RoboDK station: Assignment 3.rdk

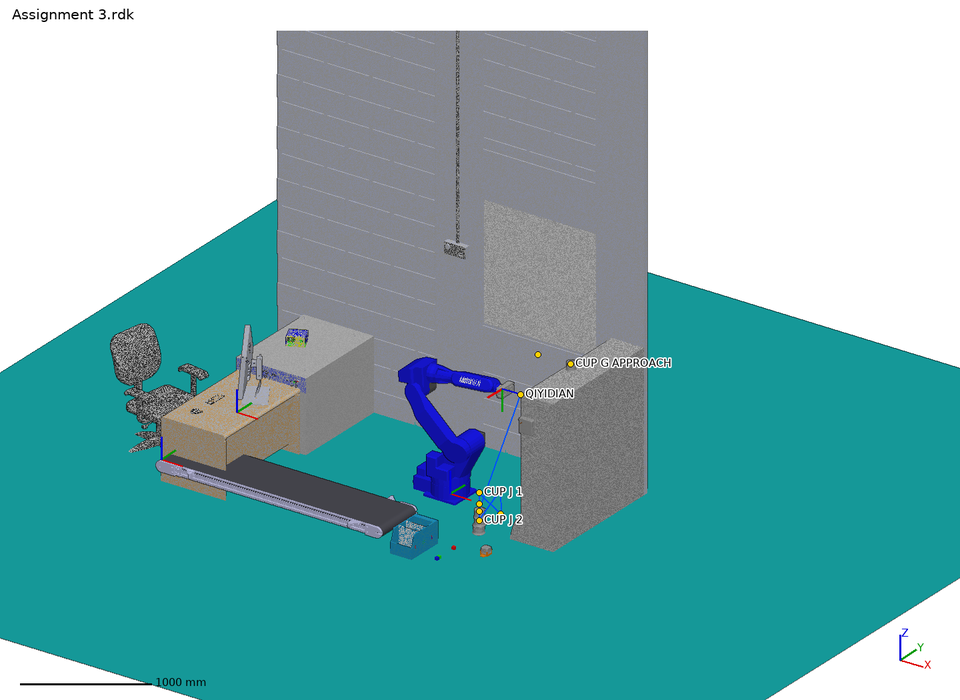
[picture v0: the station drawn from its stored meshes, robots at their saved joint values, targets as dots, program paths as lines]
Station Assignment 3 (saved by RoboDK 5.2.1). Poses are relative to the parent item; angles as X-Y-Z fixed-axis rotations.
  - frame Motoman UP6 Base at (0, 0, 0) mm
    - robot Motoman UP6: 6 axes, payload 6 kg, reach 1373 mm, repeatability 0.08 mm, weight 130 kg
        modified DH rows (alpha deg, a mm, theta deg, d mm): 0, 0, 0, 450; -90, 150, -90, 0; 0, 570, 0, 0; -90, 130, 0, 640; 90, 0, 90, 0; -90, 0, 0, 95
        joint limits [-170, -90, -82, -180, -135, -360] to [170, 155, 104, 180, 180, 360]; home [0, 0, 0, 0, 0, 0]; saved at [1.534, -46.461, -42.456, 20.981, 85.712, -117.468]
      - frame FESTO HGPL-25-60-A Base at (0, 0, 17.5) mm, rotated rx 0 ry 0 rz -6.54 deg
        - robot FESTO HGPL-25-60-A: 1 axes
            joint limits [0] to [90]; home [0]; saved at [90]
      - tool Parallel Jaw Gripper TCP, TCP at (0, 0, 187) mm, rotated rx 0 ry 0 rz -6.54 deg
  - frame Conveyor Belt Base at (-1833.5, -1202.3, 256) mm
    - robot Conveyor Belt: 1 axes
        modified DH rows (alpha deg, a mm, theta deg, d mm): 0, 0, 0, 0 linear
        base shift (0, 0, 0) mm, rotated rx 0 ry 90 rz 0 deg
        joint limits [-500000] to [500000]; home [0]; saved at [0]
      - frame Conveyor at (0, 1000, 0) mm
    - target ConveryorInf (joint target) at (50000, 0, 0) mm; joints [50000, 0, 0, 0, 0, 0] of Conveyor Belt
  - Python program Open Gripper (listed below)
  - Python program Close Gripper (listed below)
  - frame World at (0, 0, 0) mm
    - object Floor at (0, 0, 0) mm, size 8000 x 8000 x 4 mm, geometry from plane_1m.sld
    - object Collection Box at (320, -955, 0) mm, rotated rx 0 ry 0 rz -90 deg, size 350 x 201 x 200 mm, geometry from Collection Box.STEP
    - folder Cubes
      - object Red Cube at (574.85, -770.18, 12.7) mm, size 25.4 x 25.4 x 25.4 mm, geometry from box.sld
      - object Green Cube at (574.85, -970.18, 12.7) mm, size 25.4 x 25.4 x 25.4 mm, geometry from box.sld
      - object Blue Cube at (574.85, -995.58, 12.7) mm, size 25.4 x 25.4 x 25.4 mm, geometry from box.sld
    - folder Cups
      - object Cup J at (570, -430, 80) mm, rotated rx -180 ry 0 rz 0 deg, size 102.7 x 102.6 x 71.8 mm, geometry from textured.obj
        - object Room Assembly at (-1580, -795, 320) mm, rotated rx -90 ry 0 rz 90 deg, size 1945 x 4060 x 3887.6 mm, geometry from Room Assembly.STEP
        - object Cup I at (-5, 0, -65) mm, size 98.2 x 97 x 71.7 mm, geometry from textured.obj
        - object Cup H at (0.2, 1.71, -129.62) mm, size 90.9 x 92 x 71.3 mm, geometry from textured.obj
      - object Cup G at (980, 190, 1320) mm, rotated rx -180 ry 0 rz 0 deg, size 86.4 x 85.9 x 70.2 mm, geometry from textured.obj
    - object Peg at (960.21, -424.7, 1039.75) mm, size 6 x 40 x 6 mm, geometry from Peg.STEP
    - object Rubiks Cube Holder at (830, -710, 6.5) mm, rotated rx 90 ry 0 rz 90 deg, size 116 x 39.8 x 68 mm, geometry from Rubiks Cube Holder.STEP
    - object 9 Hole Peg at (977, -381, 1006) mm, rotated rx 90 ry -45 rz 0 deg, size 174.8 x 175.2 x 38.4 mm, geometry from textured.obj
    - object Rubiks Cube at (836.12, -697.93, 9.9) mm, rotated rx 0 ry 0 rz 42.55 deg, size 84.3 x 85.7 x 55.5 mm, geometry from textured.obj
    - target CUP J 1 (Cartesian target) at (570, -430, 340.32) mm, rotated rx -180 ry 0 rz 0 deg; joints [-37.03, 4.491, -44.31, 0, 48.801, 30.49] of Motoman UP6
    - target CUP J 2 (Cartesian target) at (570, -430, 105) mm, rotated rx -180 ry 0 rz 0 deg; joints [-37.03, 26.298, -46.699, 0, 72.996, 30.49] of Motoman UP6
    - target CUP I 1 (Cartesian target) at (570, -150, 250) mm, rotated rx -180 ry 0 rz 0 deg; joints [-14.744, 0.541, -59.29, 0, 59.831, 8.204] of Motoman UP6
    - target CUP I 2 (Cartesian target) at (575, -150, 50) mm, rotated rx -180 ry 0 rz 0 deg; joints [-14.621, 26.957, -57.991, 0, 84.948, 8.081] of Motoman UP6
    - target CUPJ DOWN2 (Cartesian target) at (570, -430, 181.5) mm, rotated rx -180 ry 0 rz 0 deg; joints [-37.03, 18.317, -47.056, 0, 65.374, 30.49] of Motoman UP6
    - target CUP G APPROACH (Cartesian target) at (980, 197, 1290) mm, rotated rx -90 ry 0 rz -90 deg; joints [15.761, -1.933, 11.037, 51.508, 69.694, -146.245] of Motoman UP6
    - target CUP G STOP (Cartesian target) at (680, 190, 1290) mm, rotated rx -90 ry 0 rz -90 deg; joints [25.519, -28.082, -8.487, 54.912, 58.231, -146.974] of Motoman UP6
    - target CUP G end (Cartesian target) at (570, -430, 247.55) mm, rotated rx -90 ry 0 rz -90 deg; joints [-56.187, 37.804, -62.086, -123.417, -5.484, 91.702] of Motoman UP6
    - target QIYIDIAN (Cartesian target) at (648.03, 9.8, 1017.02) mm, rotated rx -90 ry 0 rz -90 deg; joints [1.534, -46.461, -42.456, 20.981, 85.712, -117.468] of Motoman UP6
  - program Reset Objects (1 instructions, listed below)
  - Python program Initialize Objects (listed below)
  - program CUP TOWER (20 instructions, listed below)
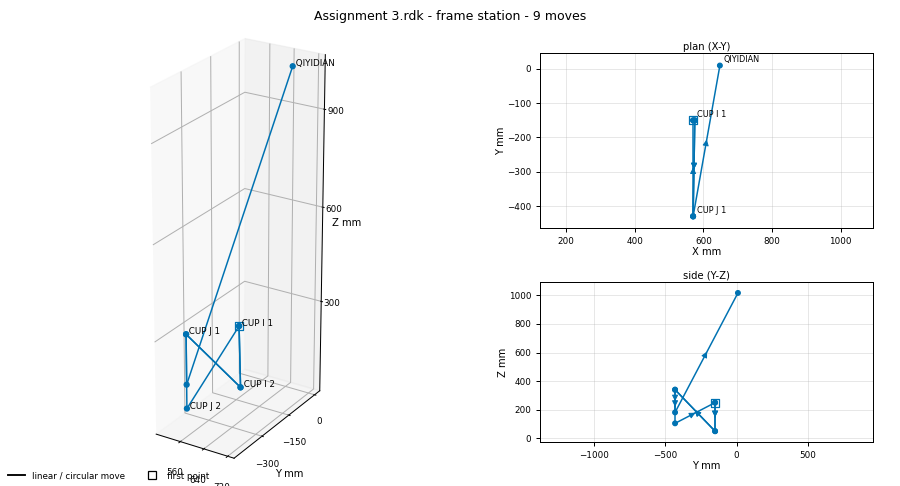
[picture p0: tool path of Assignment 3.rdk in frame station, 9 of 9 moves have a stored position in this frame; points joined in program order, loops and branches not executed]

--- Python program Open Gripper ---
from robolink import *    # RoboDK API
from robodk import *      # Robot toolbox
RDK = Robolink()

MODE = 'SIMULATION'
MODE = 'RUN_ON_ROBOT'

if MODE == 'RUN_ON_ROBOT':
    import serial
    s = serial.Serial('COM7', 9600)

gripper = RDK.Item('FESTO HGPL-25-60-A')
if gripper.Valid():
    RDK.setRunMode(RUNMODE_SIMULATE)
    gripper.MoveJ([90])
    if MODE == 'RUN_ON_ROBOT':
        RDK.setRunMode(RUNMODE_RUN_ROBOT)

time.sleep(0.5)
if MODE == 'RUN_ON_ROBOT':
    s.write(b'o')
time.sleep(0.5) #Wait for gripper to open
print('Open')

--- Python program Close Gripper ---
from robolink import *    # RoboDK API
from robodk import *      # Robot toolbox
RDK = Robolink()

MODE = 'SIMULATION'
MODE = 'RUN_ON_ROBOT'

if MODE == 'RUN_ON_ROBOT':
    import serial
    s = serial.Serial('COM7', 9600)

gripper = RDK.Item('FESTO HGPL-25-60-A')
if gripper.Valid():
    RDK.setRunMode(RUNMODE_SIMULATE)
    gripper.MoveJ([0])
    if MODE == 'RUN_ON_ROBOT':
        RDK.setRunMode(RUNMODE_RUN_ROBOT)

time.sleep(0.6)
if MODE == 'RUN_ON_ROBOT':
    s.flush()
    s.write(b'c')
time.sleep(0.5) #Wait for gripper to close
print('Closed')

--- program Reset Objects (robot Motoman UP6) ---
  Replace objects

--- Python program Initialize Objects ---
from robolink import *    # RoboDK API
from robodk import *      # Robot toolbox
RDK = Robolink()

item = RDK.Item('Cups')

world_frame = RDK.Item('World')

# Baseball
RDK.Delete(RDK.Item('Baseball'))
baseball = RDK.AddFile(RDK.getParam('PATH_OPENSTATION') + "/YCB Objects/055_baseball/tsdf/textured.obj")
baseball.setName('Baseball')
baseball.setParent(world_frame)
baseball.setPose(transl(990,0,910))

# Cups
CupFolder = RDK.Item('Cups')

RDK.Delete(RDK.Item('Cup G'))
cup_g = RDK.AddFile(RDK.getParam('PATH_OPENSTATION') + "/YCB Objects/065-g_cups/tsdf/textured.obj")
cup_g.setName('Cup G')
cup_g.setParent(CupFolder)
cup_g.setPose(transl(980,190,1320)*rotx(-pi))

RDK.Delete(RDK.Item('Cup H'))
cup_h = RDK.AddFile(RDK.getParam('PATH_OPENSTATION') + "/YCB Objects/065-h_cups/tsdf/textured.obj")
cup_h.setName('Cup H')
cup_h.setParent(CupFolder)
cup_h.setPose(transl(575.203,-151.71,78.118)*rotx(-pi))

RDK.Delete(RDK.Item('Cup I'))
cup_i = RDK.AddFile(RDK.getParam('PATH_OPENSTATION') + "/YCB Objects/065-i_cups/tsdf/textured.obj")
cup_i.setName('Cup I')
cup_i.setParent(CupFolder)
cup_i.setPose(transl(570,-150,90)*rotx(-pi))

RDK.Delete(RDK.Item('Cup J'))
cup_j = RDK.AddFile(RDK.getParam('PATH_OPENSTATION') + "/YCB Objects/065-j_cups/tsdf/textured.obj")
cup_j.setName('Cup J')
cup_j.setParent(CupFolder)
cup_j.setPose(transl(570,-430,80)*rotx(-pi))

# 9 Hole Peg
RDK.Delete(RDK.Item('9 Hole Peg'))
pegs = RDK.AddFile(RDK.getParam('PATH_OPENSTATION') + "/YCB Objects/071_nine_hole_peg_test/tsdf/textured.obj")
pegs.setName('9 Hole Peg')
pegs.setParent(world_frame)
pegs.setPose(transl(977,-381,1006)*rotx(pi/2)*rotz(pi/4))

# Rubik's cube
RDK.Delete(RDK.Item('Rubiks Cube'))
rubik = RDK.AddFile(RDK.getParam('PATH_OPENSTATION') + "/YCB Objects/077_rubiks_cube/tsdf/textured.obj")
rubik.setName('Rubiks Cube')
rubik.setParent(world_frame)
rubik.setPose(transl(836.120,-697.930,9.901)*rotz((42.550/180)*pi))

# Untextured Items
R_Cube = RDK.Item('Red Cube')
R_Cube.setPose(transl(574.847,-770.179,12.7))
G_Cube = RDK.Item('Green Cube')
G_Cube.setPose(transl(574.847,-970.179,12.7))
B_Cube = RDK.Item('Blue Cube')
B_Cube.setPose(transl(574.847,-970.179-25.4,12.7))
Rubiks_Holder = RDK.Item('Rubiks Cube Holder')
Rubiks_Holder.setPose(transl(830,-710,6.5)*roty(pi/2)*rotz(pi/2))
Pin = RDK.Item('Peg')
Pin.setPose(transl(960.212,-424.699,1039.753))

--- program CUP TOWER (robot Motoman UP6) ---
  设置参考号: World
  设置工具: Parallel Jaw Gripper TCP
  调用 Open Gripper
  MoveL (CUP I APPROACH) -> target CUP I 1
  MoveL (CUP I DOWN) -> target CUP I 2
  调用 Close Gripper
  附加到Parallel Jaw Gripper TCP
  MoveL (CUP J APPROACH) -> target CUP J 1
  MoveL (CUP J DOWN) -> target CUP J 2
  调用 Open Gripper
  分离于Parallel Jaw Gripper TCP
  MoveL (CUP I APPROACH) -> target CUP I 1
  MoveL (CUP I DOWN) -> target CUP I 2
  调用 Close Gripper
  附加到Parallel Jaw Gripper TCP
  MoveL (CUP J APPROACH) -> target CUP J 1
  MoveL (CUPJ DOWN2)
  调用 Open Gripper
  分离于Parallel Jaw Gripper TCP
  MoveL (QIYIDIAN)
